FUNCTION_BLOCK E_SR (* Basic Function Block Type *)
  (* Standard: 61499-2 *)
  (* Version 0.0, 9/12/2026, macie, Schneider Electric, Template *)
  PACKAGE Main;
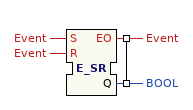
  EVENT_INPUT
    S; (* Initialization Request *)
    R; (* Normal Execution Request *)
  END_EVENT
  EVENT_OUTPUT
    EO WITH Q; (* Initialization Confirm *)
  END_EVENT
  VAR_OUTPUT
    Q : BOOL := FALSE; (* Output event qualifier *)
  END_VAR
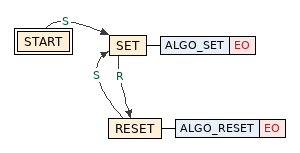
  EC_STATES
    START; (* Initial State *)
    SET : ALGO_SET -> EO; (* Initialization *)
    RESET : ALGO_RESET -> EO; (* Normal execution *)
  END_STATES
  EC_TRANSITIONS
    START TO SET := S;
    SET TO RESET := R;
    RESET TO SET := S;
  END_TRANSITIONS
  ALGORITHM ALGO_SET IN ST: (* Initialization algorithm *)
;
Q := TRUE;
  END_ALGORITHM
  ALGORITHM ALGO_RESET IN ST: (* Normally executed algorithm *)
;
Q := FALSE;
  END_ALGORITHM
END_FUNCTION_BLOCK
